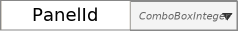
VISUALIZATION V_ApSelecCmb  // 238x31
    ComboBoxInteger (130,1 108x30), variable: VisuGVL.fbPanelImp.PanelId, text list: 'PanelCmbTxtList'
    Textfield (1,0 129x30), "PanelId"
END_VISUALIZATION

(* stored: Version 1.1.0.1, ProductVersion 3.1.4024.4
   Visu V_ApSelecCmb: Id {8188056b-7302-4217-aaf0-3dc4e25bb7d5} *)
